// TIA Portal V17 export
// export: Created 2024-09-02T12:50:22.9244543Z, ExportSetting WithDefaults, DisplayName Totally Integrated Automation Portal, DisplayVersion V17, DisplayName TIA Portal Openness, DisplayVersion V17, DisplayName TIA Portal Version Control Interface, DisplayVersion V17, DisplayName STEP 7 Professional, DisplayVersion V17, DisplayName STEP 7 Safety, DisplayVersion V17, DisplayName WinCC Professional, DisplayVersion V17
DATA_BLOCK "MdsDB2_FG01_Parameter_SLG1_OP70"   // DB912
{ S7_Optimized_Access := 'TRUE'; DB_Accessible_From_OPC_UA := 'FALSE' }
AUTHOR : OlegFuehrus
FAMILY : MOBY
NAME : MOBY
VERSION : 0.1
// stored: AutoNumber false, DBAccessibleFromOPCUA false, IsOnlyStoredInLoadMemory false, IsRetainMemResEnabled false, IsWriteProtectedInAS false, MemoryReserve 100
   VAR
      Analyze_Start : Bool;
      Analyze_Finished : Bool;
      Saving_Data_Start : Bool;
      Saveing_Data_Finished : Bool;
      Deselectionl_BEA : Array[1..8] of Bool;
      Release_BEA : Array[1..8] of Bool;
      Read_BEA : Array[1..8] of Struct
         PRG : Struct
            Dez : Int;
            _ : Array[0..15] of Bool;
         END_STRUCT;
      END_STRUCT;
      User { ExternalWritable := 'False'} : Struct
         With_Process { ExternalWritable := 'False'} : Bool;
         Lock_without_Process { ExternalWritable := 'False'} : Bool;
         In_Procecss { ExternalWritable := 'False'} : Bool;
      END_STRUCT;
   END_VAR
BEGIN
END_DATA_BLOCK
